// TIA Portal V17 export
// export: Created 2025-07-01T09:58:19.4161728Z, ExportSetting WithDefaults, DisplayName Totally Integrated Automation Portal, DisplayVersion V17 Update 8, DisplayName TIA Portal Openness, DisplayVersion V17 Update 8, DisplayName TIA Portal Version Control Interface, DisplayVersion V17, DisplayName SINAMICS Startdrive Advanced, DisplayVersion V17 SP2, DisplayName SINAMICS Startdrive G110M, G120, G120C, G120D, G120P, G115D, DisplayVersion V17 SP2, DisplayName SINAMICS Startdrive G130, G150, S120, S150, SINAMICS MV, S210, DisplayVersion V17 SP2, DisplayName STEP 7 Professional, DisplayVersion V17 Update 8, DisplayName SINUMERIK ONE STEP 7 Toolbox, DisplayVersion V17 Update 12, DisplayName SINUMERIK ONE PLC Basic Program Plus, DisplayVersion V17 Update 12, DisplayName SINUMERIK 840D sl STEP 7 Toolbox, DisplayVersion V17 Update 12, DisplayName STEP 7 Safety, DisplayVersion V17 Update 6, DisplayName WinCC Advanced, DisplayVersion V17 Update 8
FUNCTION_BLOCK "FB7001_SAFETY_DOOR"   // FB7001, LAD
{ S7_Optimized_Access := 'FALSE' }
AUTHOR : ETXETAR
VERSION : 1.0
// stored: AutoNumber false, IsIECCheckEnabled false, SetENOAutomatically false, UDAEnableTagReadback false
   VAR_INPUT
      OPTIONS_0 : Byte := 2#0000_0000;   // OPTIONS 0
      CLOSED_I : Bool;   // N.O / CLOSED INPUT
      LOCKED_I : Bool;   // N.O / LOCKED INPUT
      LOCK_CONDITIONS : Bool;   // LOCK CONDITIONS
      UNLOCK_PARTIAL_CONDITIONS : Bool;   // UNLOCK PARTIAL CONDITIONS
      HMI_REQ_LINE : Bool;   // HMI REQUEST LINE 1
      PANEL_LOCK_UNLOCK_PUSHBUTTON : Bool;   // PANEL LOCK UNLOCK PUSHBUTTON
      LOCK_AUTO_REQ : Bool;   // LOCK AUTO REQUEST
      UNLOCK_AUTO_REQ : Bool;   // UNLOCK AUTO REQUEST
      PNEUMATIC_DRIVE_UNBLOCKED : Bool;   // PNEUMATIC DRIVE 1 UNBLOCKED
   END_VAR
   VAR_OUTPUT
      NOT_CLOSED_AND_LOCKED_ALARM : Bool;   // NOT CLOSED AND LOCKED ALARM
      PNEUMATIC_DRIVE_NOT_UNBLOCKED_ALARM : Bool;   // PNEUMATIC DRIVE NOT UNBLOCKED ALARM
      NOT_OPEN_ALARM : Bool;   // NOT OPEN ALARM
      UNLOCK_REQUEST_SEOC_WRN : Bool;   // UNLOCK REQUEST SEOC WARNING
      NOT_CLOSED_WRN : Bool;   // NOT CLOSED WARNING
      HMI_MOTION_EXECUTABILITY_LEFT : Bool;   // HMI MOTION EXECUTABILITY LEFT
      HMI_MOTION_EXECUTABILITY_RIGHT : Bool;   // HMI MOTION EXECUTABILITY RIGHT
      HMI_MOTION_END_POS_LEFT : Bool;   // HMI MOTION END POSITION LEFT
      HMI_MOTION_END_POS_RIGHT : Bool;   // HMI MOTION END POSITION RIGHT
      HMI_MOTION_ACTIVE_LEFT : Bool;   // HMI MOTION ACTIVE LEFT
      HMI_MOTION_ACTIVE_RIGHT : Bool;   // HMI MOTION ACTIVE RIGHT
      UNLOCK : Bool;   // UNLOCK OUTPUT
      RED_LIGHT : Bool;   // RED LIGHT OUTPUT
      GREEN_LIGHT : Bool;   // GREEN LIGHT OUTPUT
   END_VAR
   VAR DB_SPECIFIC
      SAFETY_DOOR : "SAFETY_DOOR";
   END_VAR
   VAR_TEMP
      INPUTS_MASK : Byte;   // INPUTS_MASK
      O_BYTE_0 : Struct   // OPTIONS BYTE 0
         IMMEDIATE_STOP : Bool;   // IMMEDIATE STOP REACTION OPTION
         SEOC_WARNING : Bool;   // SEOC WARNING REACTION OPTION
         CLOSED_SENSOR : Bool;   // CLOSED SENSOR OPTION
         CIRCUIT_E2 : Bool;   // CIRCUIT E2 OPTION
         PNEUMATIC_DRIVE : Bool;   // PNEUMATIC DRIVE OPTION
         GANTRY_ROBOT_OK_TO_OPEN : Bool;   // GANTRY ROBOT OK TO OPEN SAFETY DOOR OPTION
         SPARE_6 : Bool;   // SPARE 6 OPTION
         SPARE_7 : Bool;   // SPARE 7 OPTION
      END_STRUCT;
      DB_NUMBER : DInt;   // DB NUMBER FOR ALARM AND HELP DECODING
   END_VAR
   // SAFETY_DOOR.TIMER_UNLOCK_PARTIAL_CONDITIONS.PT := T#250ms;
   // SAFETY_DOOR.TIMER_UNLOCK.PT := T#250ms;
   // SAFETY_DOOR.TIMER_PNEUMATIC_DRIVE_1_NOT_UNLOCKED.PT := T#2s;
   // SAFETY_DOOR.TIMER_NOT_OPEN.PT := T#3s;
   VAR_TEMP   // added for the SCL form of the ladder/FBD networks
      _w1 : Bool;
      _w2 : Bool;
   END_VAR
BEGIN

NETWORK
TITLE = READ INSTANCE DB
      L     DINO;
      +     10#800000;
      T     #DB_NUMBER;


REGION Network 2: OPTIONS
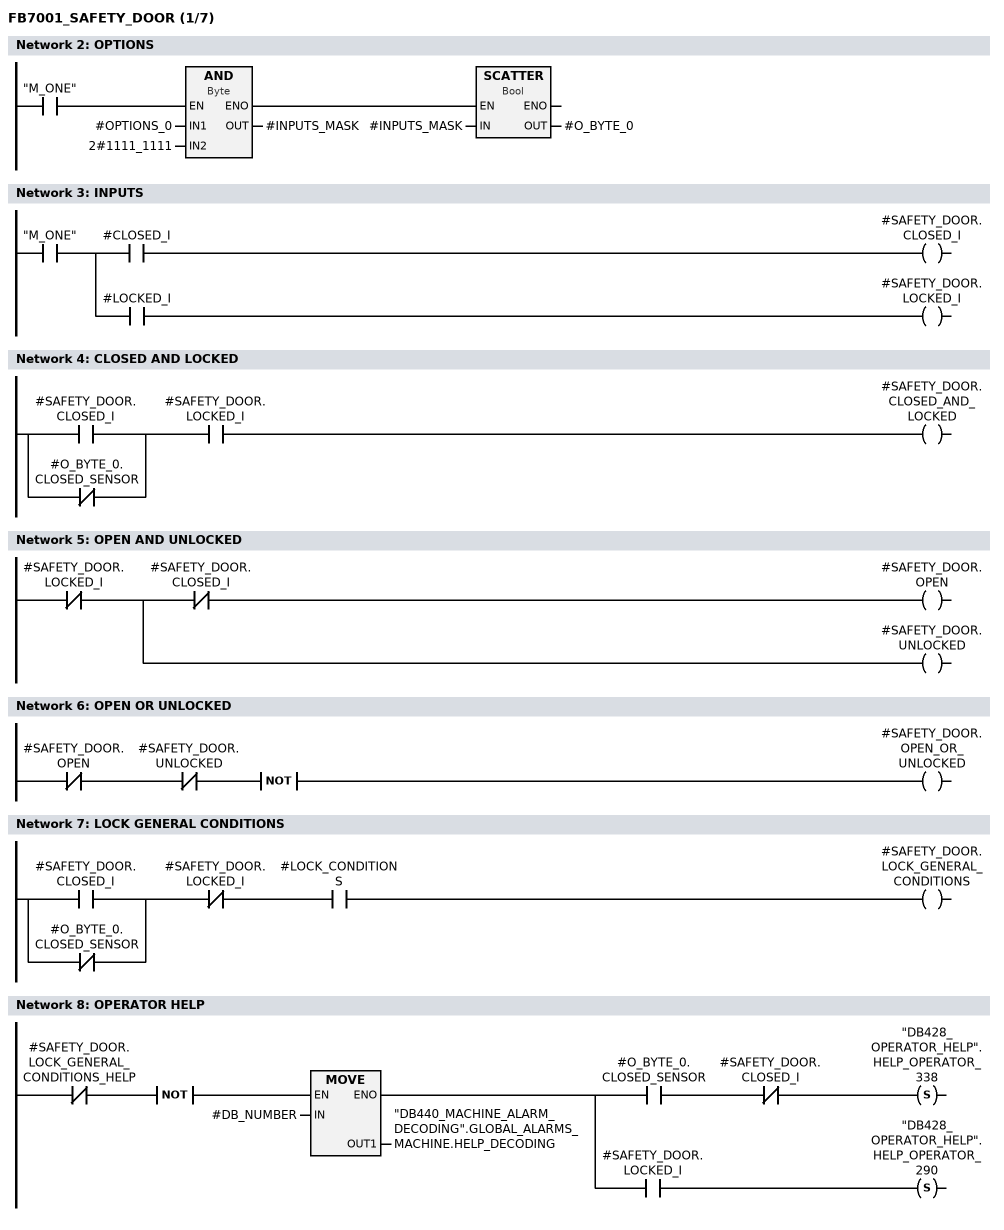
   RUNG wire#powerrail
      Contact( "M_ONE" )
      { S7_Templates := "SrcType := Byte"; S7_GenerateENO := "TRUE" } And(in1 := #OPTIONS_0, in2 := 2#1111_1111, out => #INPUTS_MASK)
      { S7_Templates := "[dest_type := Bool, src_type := Byte]" } SCATTER(IN := #INPUTS_MASK, OUT => #O_BYTE_0)
   END_RUNG
   // the same network as SCL:
   IF "M_ONE" THEN
       #INPUTS_MASK := #OPTIONS_0 AND 2#1111_1111;
       SCATTER(IN := #INPUTS_MASK, OUT => #O_BYTE_0);
   END_IF;
END_REGION

REGION Network 3: INPUTS
   RUNG wire#powerrail
      Contact( "M_ONE" )
      wire#w1
      Contact( #CLOSED_I )
      Coil( #SAFETY_DOOR.CLOSED_I )
   END_RUNG
   RUNG wire#w1
      Contact( #LOCKED_I )
      Coil( #SAFETY_DOOR.LOCKED_I )
   END_RUNG
   // the same network as SCL:
   #SAFETY_DOOR.CLOSED_I := "M_ONE" AND #CLOSED_I;
   #SAFETY_DOOR.LOCKED_I := "M_ONE" AND #LOCKED_I;
END_REGION

REGION Network 4: CLOSED AND LOCKED
   RUNG wire#powerrail
      Contact( #SAFETY_DOOR.CLOSED_I )
      wire#w1
      Contact( #SAFETY_DOOR.LOCKED_I )
      Coil( #SAFETY_DOOR.CLOSED_AND_LOCKED )
   END_RUNG
   RUNG wire#powerrail
      I_Contact( #O_BYTE_0.CLOSED_SENSOR )
   END_RUNG wire#w1
   // the same network as SCL:
   #SAFETY_DOOR.CLOSED_AND_LOCKED := (#SAFETY_DOOR.CLOSED_I OR NOT #O_BYTE_0.CLOSED_SENSOR) AND #SAFETY_DOOR.LOCKED_I;
END_REGION

REGION Network 5: OPEN AND UNLOCKED
   RUNG wire#powerrail
      I_Contact( #SAFETY_DOOR.LOCKED_I )
      wire#w1
      I_Contact( #SAFETY_DOOR.CLOSED_I )
      Coil( #SAFETY_DOOR.OPEN )
   END_RUNG
   RUNG wire#w1
      Coil( #SAFETY_DOOR.UNLOCKED )
   END_RUNG
   // the same network as SCL:
   #_w1 := NOT #SAFETY_DOOR.LOCKED_I;
   #SAFETY_DOOR.OPEN := #_w1 AND NOT #SAFETY_DOOR.CLOSED_I;
   #SAFETY_DOOR.UNLOCKED := #_w1;
END_REGION

REGION Network 6: OPEN OR UNLOCKED
   RUNG wire#powerrail
      I_Contact( #SAFETY_DOOR.OPEN )
      I_Contact( #SAFETY_DOOR.UNLOCKED )
      Not()
      Coil( #SAFETY_DOOR.OPEN_OR_UNLOCKED )
   END_RUNG
   // the same network as SCL:
   #SAFETY_DOOR.OPEN_OR_UNLOCKED := NOT (NOT #SAFETY_DOOR.OPEN AND NOT #SAFETY_DOOR.UNLOCKED);
END_REGION

REGION Network 7: LOCK GENERAL CONDITIONS
   RUNG wire#powerrail
      Contact( #SAFETY_DOOR.CLOSED_I )
      wire#w1
      I_Contact( #SAFETY_DOOR.LOCKED_I )
      Contact( #LOCK_CONDITIONS )
      Coil( #SAFETY_DOOR.LOCK_GENERAL_CONDITIONS )
   END_RUNG
   RUNG wire#powerrail
      I_Contact( #O_BYTE_0.CLOSED_SENSOR )
   END_RUNG wire#w1
   // the same network as SCL:
   #SAFETY_DOOR.LOCK_GENERAL_CONDITIONS := (#SAFETY_DOOR.CLOSED_I OR NOT #O_BYTE_0.CLOSED_SENSOR) AND NOT #SAFETY_DOOR.LOCKED_I AND #LOCK_CONDITIONS;
END_REGION

REGION Network 8: OPERATOR HELP
   RUNG wire#powerrail
      I_Contact( #SAFETY_DOOR.LOCK_GENERAL_CONDITIONS_HELP )
      Not()
      { S7_GenerateENO := "TRUE" } Move(in := #DB_NUMBER, out1 => "DB440_MACHINE_ALARM_DECODING".GLOBAL_ALARMS_MACHINE.HELP_DECODING)
      wire#w1
      Contact( #O_BYTE_0.CLOSED_SENSOR )
      I_Contact( #SAFETY_DOOR.CLOSED_I )
      S_Coil( "DB428_OPERATOR_HELP".HELP_OPERATOR_338 )
   END_RUNG
   RUNG wire#w1
      Contact( #SAFETY_DOOR.LOCKED_I )
      S_Coil( "DB428_OPERATOR_HELP".HELP_OPERATOR_290 )
   END_RUNG
   // the same network as SCL:
   // ENO of a box is taken as its EN; it also drops when the box reports an error
   #_w1 := NOT (NOT #SAFETY_DOOR.LOCK_GENERAL_CONDITIONS_HELP);
   IF #_w1 THEN "DB440_MACHINE_ALARM_DECODING".GLOBAL_ALARMS_MACHINE.HELP_DECODING := #DB_NUMBER; END_IF;
   IF #_w1 AND #O_BYTE_0.CLOSED_SENSOR AND NOT #SAFETY_DOOR.CLOSED_I THEN
       "DB428_OPERATOR_HELP".HELP_OPERATOR_338 := TRUE;
   END_IF;
   IF #_w1 AND #SAFETY_DOOR.LOCKED_I THEN "DB428_OPERATOR_HELP".HELP_OPERATOR_290 := TRUE; END_IF;
END_REGION

REGION Network 9: LOCK MANUAL REQUEST
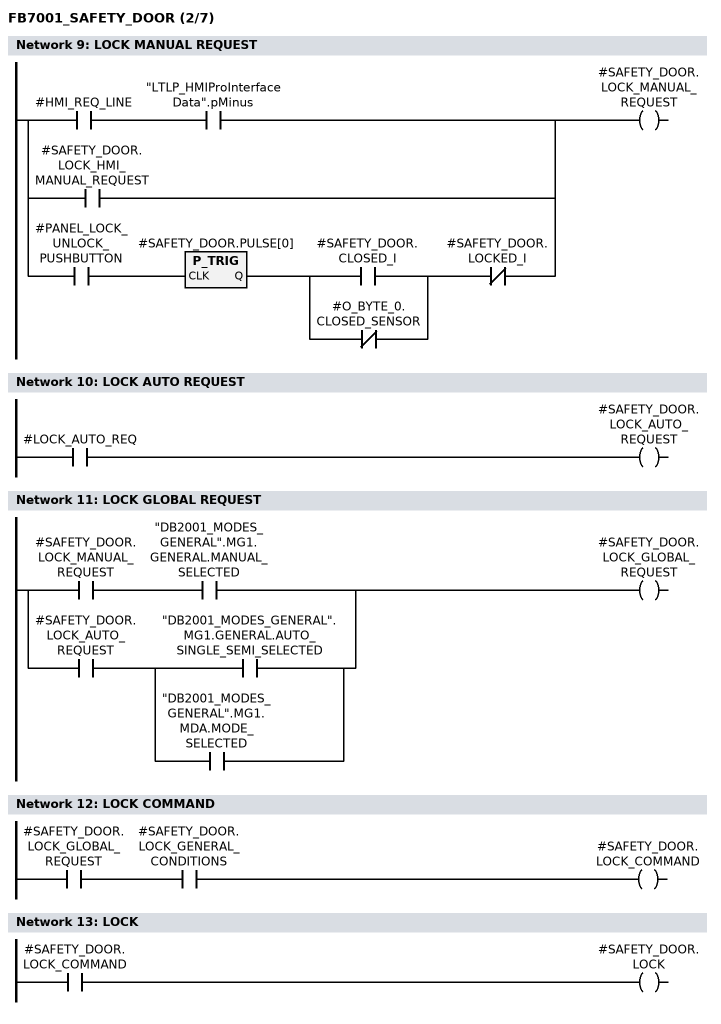
   RUNG wire#powerrail
      Contact( #HMI_REQ_LINE )
      Contact( "LTLP_HMIProInterfaceData".pMinus )
      wire#w1
      Coil( #SAFETY_DOOR.LOCK_MANUAL_REQUEST )
   END_RUNG
   RUNG wire#powerrail
      Contact( #SAFETY_DOOR.LOCK_HMI_MANUAL_REQUEST )
   END_RUNG wire#w1
   RUNG wire#powerrail
      Contact( #PANEL_LOCK_UNLOCK_PUSHBUTTON )
      P_Trig( #SAFETY_DOOR.PULSE[0] )
      wire#w2
      Contact( #SAFETY_DOOR.CLOSED_I )
      wire#w3
      I_Contact( #SAFETY_DOOR.LOCKED_I )
   END_RUNG wire#w1
   RUNG wire#w2
      I_Contact( #O_BYTE_0.CLOSED_SENSOR )
   END_RUNG wire#w3
   // the same network as SCL:
   #_w1 := #PANEL_LOCK_UNLOCK_PUSHBUTTON AND NOT #SAFETY_DOOR.PULSE[0];   // rising edge
   #SAFETY_DOOR.PULSE[0] := #PANEL_LOCK_UNLOCK_PUSHBUTTON;
   #SAFETY_DOOR.LOCK_MANUAL_REQUEST := (#HMI_REQ_LINE AND "LTLP_HMIProInterfaceData".pMinus) OR #SAFETY_DOOR.LOCK_HMI_MANUAL_REQUEST OR (#_w1 AND (#SAFETY_DOOR.CLOSED_I OR NOT #O_BYTE_0.CLOSED_SENSOR) AND NOT #SAFETY_DOOR.LOCKED_I);
END_REGION

REGION Network 10: LOCK AUTO REQUEST
   RUNG wire#powerrail
      Contact( #LOCK_AUTO_REQ )
      Coil( #SAFETY_DOOR.LOCK_AUTO_REQUEST )
   END_RUNG
   // the same network as SCL:
   #SAFETY_DOOR.LOCK_AUTO_REQUEST := #LOCK_AUTO_REQ;
END_REGION

REGION Network 11: LOCK GLOBAL REQUEST
   RUNG wire#powerrail
      Contact( #SAFETY_DOOR.LOCK_MANUAL_REQUEST )
      Contact( "DB2001_MODES_GENERAL".MG1.GENERAL.MANUAL_SELECTED )
      wire#w1
      Coil( #SAFETY_DOOR.LOCK_GLOBAL_REQUEST )
   END_RUNG
   RUNG wire#powerrail
      Contact( #SAFETY_DOOR.LOCK_AUTO_REQUEST )
      wire#w2
      Contact( "DB2001_MODES_GENERAL".MG1.GENERAL.AUTO_SINGLE_SEMI_SELECTED )
   END_RUNG wire#w1
   RUNG wire#w2
      Contact( "DB2001_MODES_GENERAL".MG1.MDA.MODE_SELECTED )
   END_RUNG wire#w1
   // the same network as SCL:
   #SAFETY_DOOR.LOCK_GLOBAL_REQUEST := (#SAFETY_DOOR.LOCK_MANUAL_REQUEST AND "DB2001_MODES_GENERAL".MG1.GENERAL.MANUAL_SELECTED) OR (#SAFETY_DOOR.LOCK_AUTO_REQUEST AND ("DB2001_MODES_GENERAL".MG1.GENERAL.AUTO_SINGLE_SEMI_SELECTED OR "DB2001_MODES_GENERAL".MG1.MDA.MODE_SELECTED));
END_REGION

REGION Network 12: LOCK COMMAND
   RUNG wire#powerrail
      Contact( #SAFETY_DOOR.LOCK_GLOBAL_REQUEST )
      Contact( #SAFETY_DOOR.LOCK_GENERAL_CONDITIONS )
      Coil( #SAFETY_DOOR.LOCK_COMMAND )
   END_RUNG
   // the same network as SCL:
   #SAFETY_DOOR.LOCK_COMMAND := #SAFETY_DOOR.LOCK_GLOBAL_REQUEST AND #SAFETY_DOOR.LOCK_GENERAL_CONDITIONS;
END_REGION

REGION Network 13: LOCK
   RUNG wire#powerrail
      Contact( #SAFETY_DOOR.LOCK_COMMAND )
      Coil( #SAFETY_DOOR.LOCK )
   END_RUNG
   // the same network as SCL:
   #SAFETY_DOOR.LOCK := #SAFETY_DOOR.LOCK_COMMAND;
END_REGION

REGION Network 14: UNLOCK PARTIAL CONDITIONS AUXILIARY
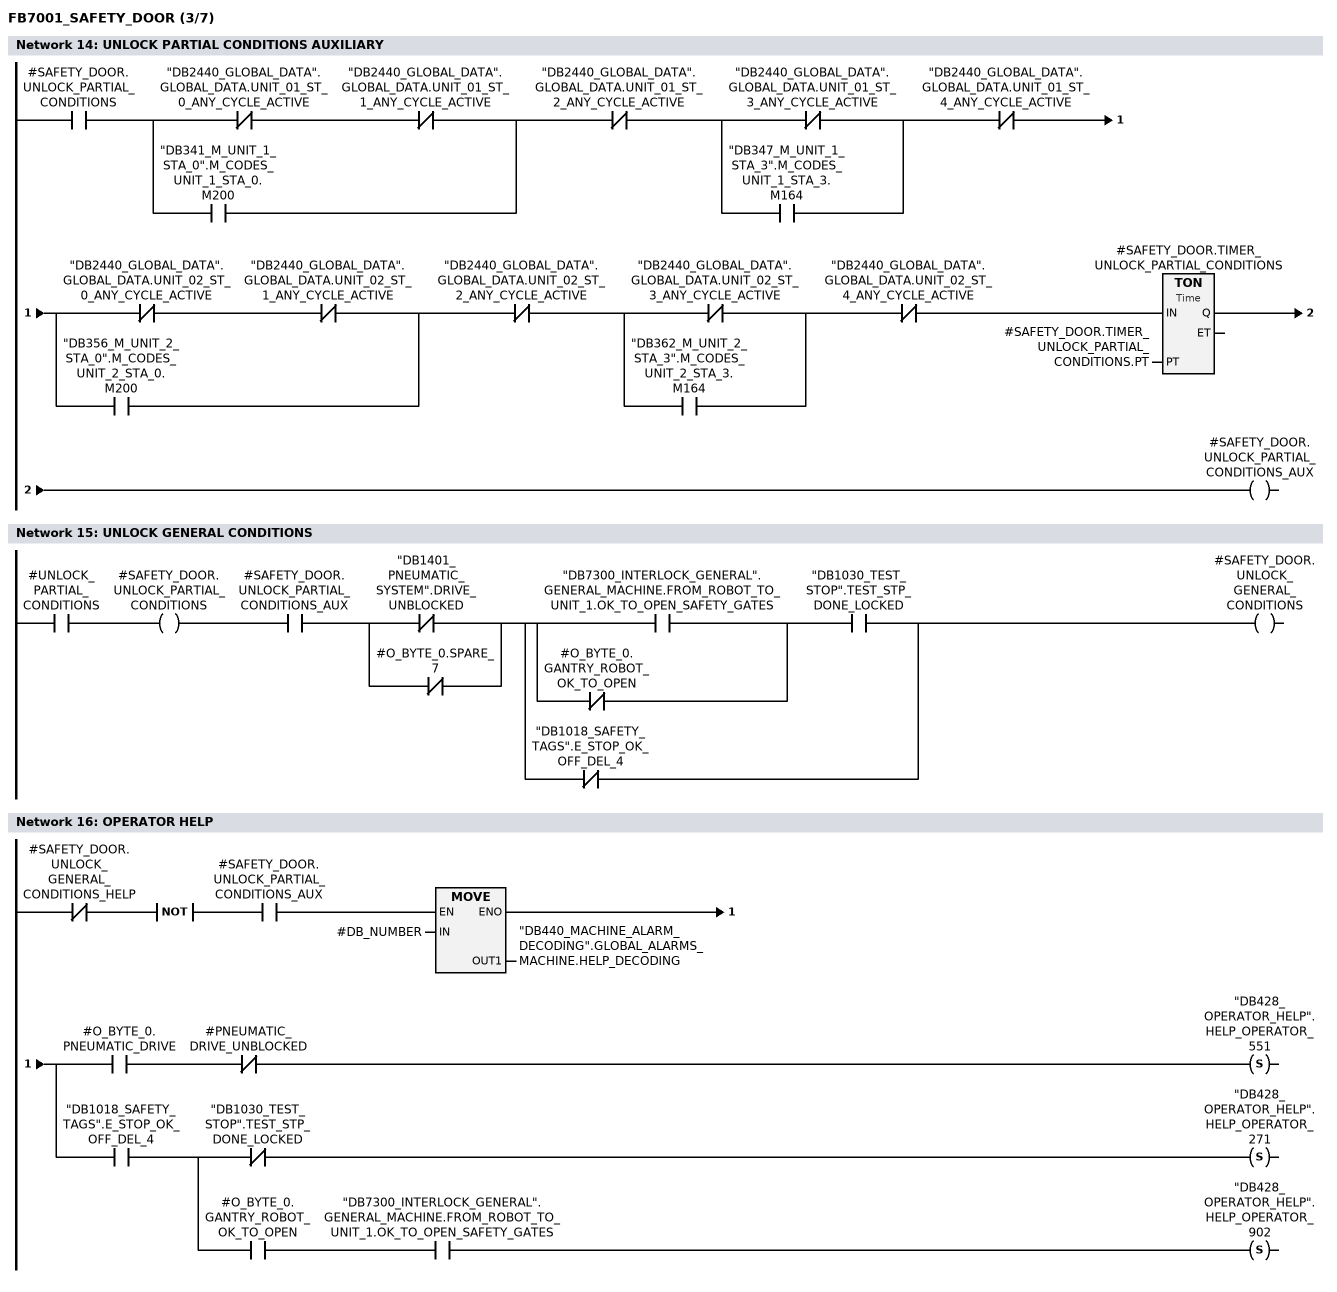
   RUNG wire#powerrail
      Contact( #SAFETY_DOOR.UNLOCK_PARTIAL_CONDITIONS )
      wire#w1
      I_Contact( "DB2440_GLOBAL_DATA".GLOBAL_DATA.UNIT_01_ST_0_ANY_CYCLE_ACTIVE )
      I_Contact( "DB2440_GLOBAL_DATA".GLOBAL_DATA.UNIT_01_ST_1_ANY_CYCLE_ACTIVE )
      wire#w2
      I_Contact( "DB2440_GLOBAL_DATA".GLOBAL_DATA.UNIT_01_ST_2_ANY_CYCLE_ACTIVE )
      wire#w3
      I_Contact( "DB2440_GLOBAL_DATA".GLOBAL_DATA.UNIT_01_ST_3_ANY_CYCLE_ACTIVE )
      wire#w4
      I_Contact( "DB2440_GLOBAL_DATA".GLOBAL_DATA.UNIT_01_ST_4_ANY_CYCLE_ACTIVE )
      wire#w5
      I_Contact( "DB2440_GLOBAL_DATA".GLOBAL_DATA.UNIT_02_ST_0_ANY_CYCLE_ACTIVE )
      I_Contact( "DB2440_GLOBAL_DATA".GLOBAL_DATA.UNIT_02_ST_1_ANY_CYCLE_ACTIVE )
      wire#w6
      I_Contact( "DB2440_GLOBAL_DATA".GLOBAL_DATA.UNIT_02_ST_2_ANY_CYCLE_ACTIVE )
      wire#w7
      I_Contact( "DB2440_GLOBAL_DATA".GLOBAL_DATA.UNIT_02_ST_3_ANY_CYCLE_ACTIVE )
      wire#w8
      I_Contact( "DB2440_GLOBAL_DATA".GLOBAL_DATA.UNIT_02_ST_4_ANY_CYCLE_ACTIVE )
      { S7_Templates := "time_type := Time" } #SAFETY_DOOR.TIMER_UNLOCK_PARTIAL_CONDITIONS.TON(pt := #SAFETY_DOOR.TIMER_UNLOCK_PARTIAL_CONDITIONS.PT, et =>)
      Coil( #SAFETY_DOOR.UNLOCK_PARTIAL_CONDITIONS_AUX )
   END_RUNG
   RUNG wire#w1
      Contact( "DB341_M_UNIT_1_STA_0".M_CODES_UNIT_1_STA_0.M200 )
   END_RUNG wire#w2
   RUNG wire#w3
      Contact( "DB347_M_UNIT_1_STA_3".M_CODES_UNIT_1_STA_3.M164 )
   END_RUNG wire#w4
   RUNG wire#w5
      Contact( "DB356_M_UNIT_2_STA_0".M_CODES_UNIT_2_STA_0.M200 )
   END_RUNG wire#w6
   RUNG wire#w7
      Contact( "DB362_M_UNIT_2_STA_3".M_CODES_UNIT_2_STA_3.M164 )
   END_RUNG wire#w8
   // the same network as SCL:
   #SAFETY_DOOR.TIMER_UNLOCK_PARTIAL_CONDITIONS.TON(IN := #SAFETY_DOOR.UNLOCK_PARTIAL_CONDITIONS AND ((NOT "DB2440_GLOBAL_DATA".GLOBAL_DATA.UNIT_01_ST_0_ANY_CYCLE_ACTIVE AND NOT "DB2440_GLOBAL_DATA".GLOBAL_DATA.UNIT_01_ST_1_ANY_CYCLE_ACTIVE) OR "DB341_M_UNIT_1_STA_0".M_CODES_UNIT_1_STA_0.M200) AND NOT "DB2440_GLOBAL_DATA".GLOBAL_DATA.UNIT_01_ST_2_ANY_CYCLE_ACTIVE AND (NOT "DB2440_GLOBAL_DATA".GLOBAL_DATA.UNIT_01_ST_3_ANY_CYCLE_ACTIVE OR "DB347_M_UNIT_1_STA_3".M_CODES_UNIT_1_STA_3.M164) AND NOT "DB2440_GLOBAL_DATA".GLOBAL_DATA.UNIT_01_ST_4_ANY_CYCLE_ACTIVE AND ((NOT "DB2440_GLOBAL_DATA".GLOBAL_DATA.UNIT_02_ST_0_ANY_CYCLE_ACTIVE AND NOT "DB2440_GLOBAL_DATA".GLOBAL_DATA.UNIT_02_ST_1_ANY_CYCLE_ACTIVE) OR "DB356_M_UNIT_2_STA_0".M_CODES_UNIT_2_STA_0.M200) AND NOT "DB2440_GLOBAL_DATA".GLOBAL_DATA.UNIT_02_ST_2_ANY_CYCLE_ACTIVE AND (NOT "DB2440_GLOBAL_DATA".GLOBAL_DATA.UNIT_02_ST_3_ANY_CYCLE_ACTIVE OR "DB362_M_UNIT_2_STA_3".M_CODES_UNIT_2_STA_3.M164) AND NOT "DB2440_GLOBAL_DATA".GLOBAL_DATA.UNIT_02_ST_4_ANY_CYCLE_ACTIVE,
                           PT := #SAFETY_DOOR.TIMER_UNLOCK_PARTIAL_CONDITIONS.PT);
   #SAFETY_DOOR.UNLOCK_PARTIAL_CONDITIONS_AUX := #SAFETY_DOOR.TIMER_UNLOCK_PARTIAL_CONDITIONS.Q;
END_REGION

REGION Network 15: UNLOCK GENERAL CONDITIONS
   RUNG wire#powerrail
      Contact( #UNLOCK_PARTIAL_CONDITIONS )
      Coil( #SAFETY_DOOR.UNLOCK_PARTIAL_CONDITIONS )
      Contact( #SAFETY_DOOR.UNLOCK_PARTIAL_CONDITIONS_AUX )
      wire#w1
      I_Contact( "DB1401_PNEUMATIC_SYSTEM".DRIVE_UNBLOCKED )
      wire#w2
      Contact( "DB7300_INTERLOCK_GENERAL".GENERAL_MACHINE.FROM_ROBOT_TO_UNIT_1.OK_TO_OPEN_SAFETY_GATES )
      wire#w3
      Contact( "DB1030_TEST_STOP".TEST_STP_DONE_LOCKED )
      wire#w4
      Coil( #SAFETY_DOOR.UNLOCK_GENERAL_CONDITIONS )
   END_RUNG
   RUNG wire#w1
      I_Contact( #O_BYTE_0.SPARE_7 )
   END_RUNG wire#w2
   RUNG wire#w2
      I_Contact( #O_BYTE_0.GANTRY_ROBOT_OK_TO_OPEN )
   END_RUNG wire#w3
   RUNG wire#w2
      I_Contact( "DB1018_SAFETY_TAGS".E_STOP_OK_OFF_DEL_4 )
   END_RUNG wire#w4
   // the same network as SCL:
   #SAFETY_DOOR.UNLOCK_PARTIAL_CONDITIONS := #UNLOCK_PARTIAL_CONDITIONS;
   #SAFETY_DOOR.UNLOCK_GENERAL_CONDITIONS := #UNLOCK_PARTIAL_CONDITIONS AND #SAFETY_DOOR.UNLOCK_PARTIAL_CONDITIONS_AUX AND (NOT "DB1401_PNEUMATIC_SYSTEM".DRIVE_UNBLOCKED OR NOT #O_BYTE_0.SPARE_7) AND ((("DB7300_INTERLOCK_GENERAL".GENERAL_MACHINE.FROM_ROBOT_TO_UNIT_1.OK_TO_OPEN_SAFETY_GATES OR NOT #O_BYTE_0.GANTRY_ROBOT_OK_TO_OPEN) AND "DB1030_TEST_STOP".TEST_STP_DONE_LOCKED) OR NOT "DB1018_SAFETY_TAGS".E_STOP_OK_OFF_DEL_4);
END_REGION

REGION Network 16: OPERATOR HELP
   RUNG wire#powerrail
      I_Contact( #SAFETY_DOOR.UNLOCK_GENERAL_CONDITIONS_HELP )
      Not()
      Contact( #SAFETY_DOOR.UNLOCK_PARTIAL_CONDITIONS_AUX )
      { S7_GenerateENO := "TRUE" } Move(in := #DB_NUMBER, out1 => "DB440_MACHINE_ALARM_DECODING".GLOBAL_ALARMS_MACHINE.HELP_DECODING)
      wire#w1
      Contact( #O_BYTE_0.PNEUMATIC_DRIVE )
      I_Contact( #PNEUMATIC_DRIVE_UNBLOCKED )
      S_Coil( "DB428_OPERATOR_HELP".HELP_OPERATOR_551 )
   END_RUNG
   RUNG wire#w1
      Contact( "DB1018_SAFETY_TAGS".E_STOP_OK_OFF_DEL_4 )
      wire#w2
      I_Contact( "DB1030_TEST_STOP".TEST_STP_DONE_LOCKED )
      S_Coil( "DB428_OPERATOR_HELP".HELP_OPERATOR_271 )
   END_RUNG
   RUNG wire#w2
      Contact( #O_BYTE_0.GANTRY_ROBOT_OK_TO_OPEN )
      Contact( "DB7300_INTERLOCK_GENERAL".GENERAL_MACHINE.FROM_ROBOT_TO_UNIT_1.OK_TO_OPEN_SAFETY_GATES )
      S_Coil( "DB428_OPERATOR_HELP".HELP_OPERATOR_902 )
   END_RUNG
   // the same network as SCL:
   // ENO of a box is taken as its EN; it also drops when the box reports an error
   #_w1 := NOT (NOT #SAFETY_DOOR.UNLOCK_GENERAL_CONDITIONS_HELP) AND #SAFETY_DOOR.UNLOCK_PARTIAL_CONDITIONS_AUX;
   IF #_w1 THEN "DB440_MACHINE_ALARM_DECODING".GLOBAL_ALARMS_MACHINE.HELP_DECODING := #DB_NUMBER; END_IF;
   IF #_w1 AND #O_BYTE_0.PNEUMATIC_DRIVE AND NOT #PNEUMATIC_DRIVE_UNBLOCKED THEN
       "DB428_OPERATOR_HELP".HELP_OPERATOR_551 := TRUE;
   END_IF;
   #_w2 := #_w1 AND "DB1018_SAFETY_TAGS".E_STOP_OK_OFF_DEL_4;
   IF #_w2 AND NOT "DB1030_TEST_STOP".TEST_STP_DONE_LOCKED THEN
       "DB428_OPERATOR_HELP".HELP_OPERATOR_271 := TRUE;
   END_IF;
   IF #_w2 AND #O_BYTE_0.GANTRY_ROBOT_OK_TO_OPEN AND "DB7300_INTERLOCK_GENERAL".GENERAL_MACHINE.FROM_ROBOT_TO_UNIT_1.OK_TO_OPEN_SAFETY_GATES THEN
       "DB428_OPERATOR_HELP".HELP_OPERATOR_902 := TRUE;
   END_IF;
END_REGION

REGION Network 17: UNLOCK MANUAL REQUEST
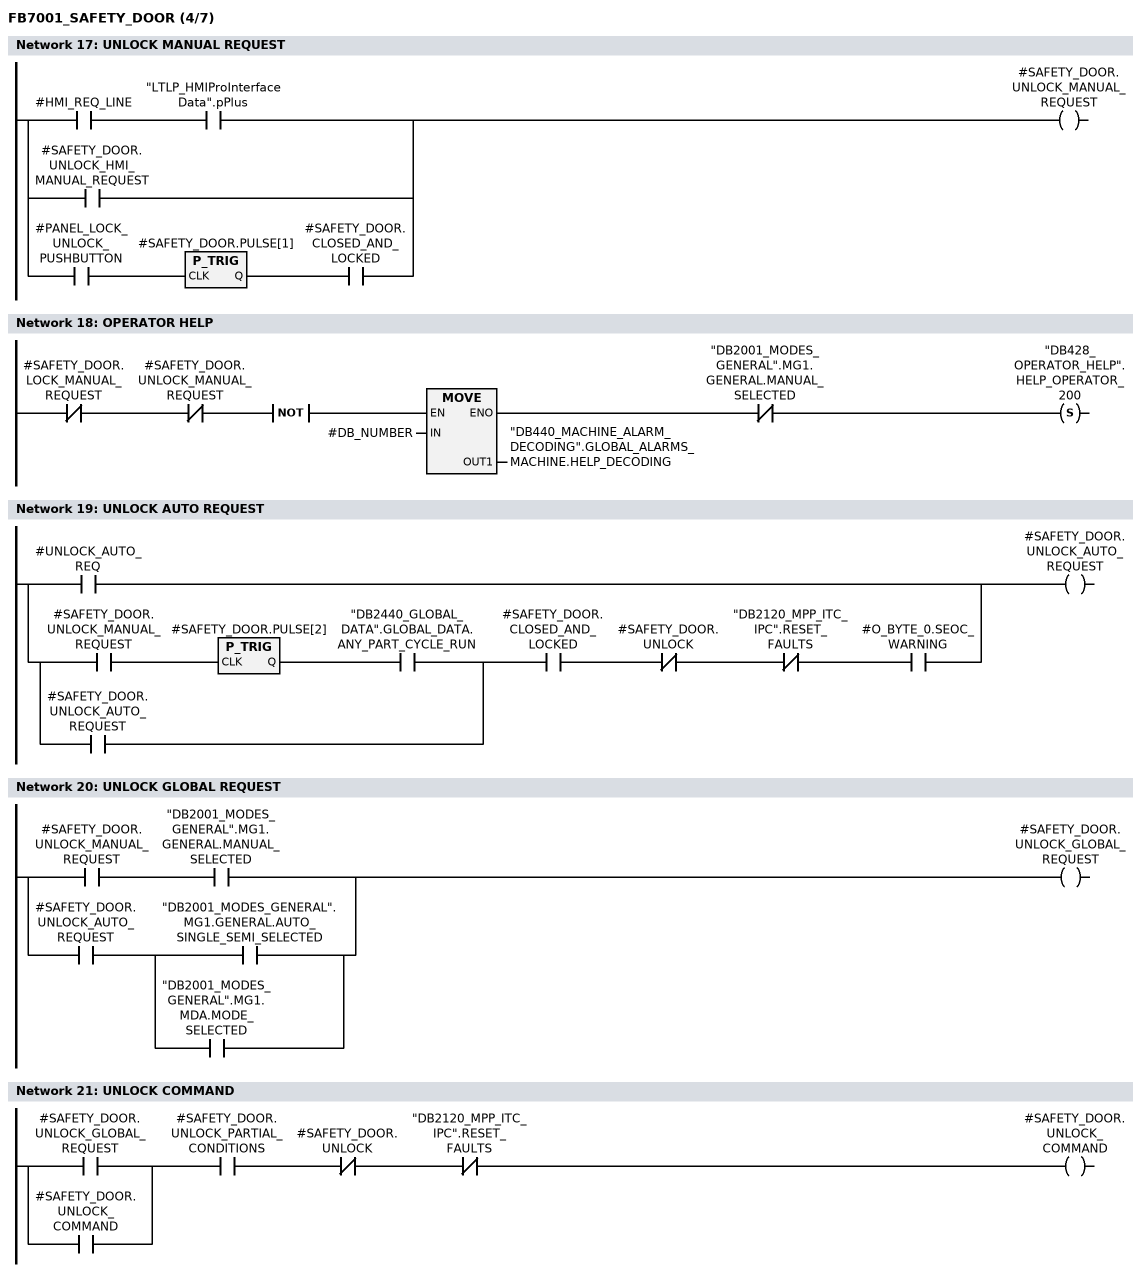
   RUNG wire#powerrail
      Contact( #HMI_REQ_LINE )
      Contact( "LTLP_HMIProInterfaceData".pPlus )
      wire#w1
      Coil( #SAFETY_DOOR.UNLOCK_MANUAL_REQUEST )
   END_RUNG
   RUNG wire#powerrail
      Contact( #SAFETY_DOOR.UNLOCK_HMI_MANUAL_REQUEST )
   END_RUNG wire#w1
   RUNG wire#powerrail
      Contact( #PANEL_LOCK_UNLOCK_PUSHBUTTON )
      P_Trig( #SAFETY_DOOR.PULSE[1] )
      Contact( #SAFETY_DOOR.CLOSED_AND_LOCKED )
   END_RUNG wire#w1
   // the same network as SCL:
   #_w1 := #PANEL_LOCK_UNLOCK_PUSHBUTTON AND NOT #SAFETY_DOOR.PULSE[1];   // rising edge
   #SAFETY_DOOR.PULSE[1] := #PANEL_LOCK_UNLOCK_PUSHBUTTON;
   #SAFETY_DOOR.UNLOCK_MANUAL_REQUEST := (#HMI_REQ_LINE AND "LTLP_HMIProInterfaceData".pPlus) OR #SAFETY_DOOR.UNLOCK_HMI_MANUAL_REQUEST OR (#_w1 AND #SAFETY_DOOR.CLOSED_AND_LOCKED);
END_REGION

REGION Network 18: OPERATOR HELP
   RUNG wire#powerrail
      I_Contact( #SAFETY_DOOR.LOCK_MANUAL_REQUEST )
      I_Contact( #SAFETY_DOOR.UNLOCK_MANUAL_REQUEST )
      Not()
      { S7_GenerateENO := "TRUE" } Move(in := #DB_NUMBER, out1 => "DB440_MACHINE_ALARM_DECODING".GLOBAL_ALARMS_MACHINE.HELP_DECODING)
      I_Contact( "DB2001_MODES_GENERAL".MG1.GENERAL.MANUAL_SELECTED )
      S_Coil( "DB428_OPERATOR_HELP".HELP_OPERATOR_200 )
   END_RUNG
   // the same network as SCL:
   // ENO of a box is taken as its EN; it also drops when the box reports an error
   #_w1 := NOT (NOT #SAFETY_DOOR.LOCK_MANUAL_REQUEST AND NOT #SAFETY_DOOR.UNLOCK_MANUAL_REQUEST);
   IF #_w1 THEN "DB440_MACHINE_ALARM_DECODING".GLOBAL_ALARMS_MACHINE.HELP_DECODING := #DB_NUMBER; END_IF;
   IF #_w1 AND NOT "DB2001_MODES_GENERAL".MG1.GENERAL.MANUAL_SELECTED THEN
       "DB428_OPERATOR_HELP".HELP_OPERATOR_200 := TRUE;
   END_IF;
END_REGION

REGION Network 19: UNLOCK AUTO REQUEST
   RUNG wire#powerrail
      Contact( #UNLOCK_AUTO_REQ )
      wire#w1
      Coil( #SAFETY_DOOR.UNLOCK_AUTO_REQUEST )
   END_RUNG
   RUNG wire#powerrail
      Contact( #SAFETY_DOOR.UNLOCK_MANUAL_REQUEST )
      P_Trig( #SAFETY_DOOR.PULSE[2] )
      Contact( "DB2440_GLOBAL_DATA".GLOBAL_DATA.ANY_PART_CYCLE_RUN )
      wire#w2
      Contact( #SAFETY_DOOR.CLOSED_AND_LOCKED )
      I_Contact( #SAFETY_DOOR.UNLOCK )
      I_Contact( "DB2120_MPP_ITC_IPC".RESET_FAULTS )
      Contact( #O_BYTE_0.SEOC_WARNING )
   END_RUNG wire#w1
   RUNG wire#powerrail
      Contact( #SAFETY_DOOR.UNLOCK_AUTO_REQUEST )
   END_RUNG wire#w2
   // the same network as SCL:
   #_w1 := #SAFETY_DOOR.UNLOCK_MANUAL_REQUEST AND NOT #SAFETY_DOOR.PULSE[2];   // rising edge
   #SAFETY_DOOR.PULSE[2] := #SAFETY_DOOR.UNLOCK_MANUAL_REQUEST;
   #SAFETY_DOOR.UNLOCK_AUTO_REQUEST := #UNLOCK_AUTO_REQ OR (((#_w1 AND "DB2440_GLOBAL_DATA".GLOBAL_DATA.ANY_PART_CYCLE_RUN) OR #SAFETY_DOOR.UNLOCK_AUTO_REQUEST) AND #SAFETY_DOOR.CLOSED_AND_LOCKED AND NOT #SAFETY_DOOR.UNLOCK AND NOT "DB2120_MPP_ITC_IPC".RESET_FAULTS AND #O_BYTE_0.SEOC_WARNING);
END_REGION

REGION Network 20: UNLOCK GLOBAL REQUEST
   RUNG wire#powerrail
      Contact( #SAFETY_DOOR.UNLOCK_MANUAL_REQUEST )
      Contact( "DB2001_MODES_GENERAL".MG1.GENERAL.MANUAL_SELECTED )
      wire#w1
      Coil( #SAFETY_DOOR.UNLOCK_GLOBAL_REQUEST )
   END_RUNG
   RUNG wire#powerrail
      Contact( #SAFETY_DOOR.UNLOCK_AUTO_REQUEST )
      wire#w2
      Contact( "DB2001_MODES_GENERAL".MG1.GENERAL.AUTO_SINGLE_SEMI_SELECTED )
   END_RUNG wire#w1
   RUNG wire#w2
      Contact( "DB2001_MODES_GENERAL".MG1.MDA.MODE_SELECTED )
   END_RUNG wire#w1
   // the same network as SCL:
   #SAFETY_DOOR.UNLOCK_GLOBAL_REQUEST := (#SAFETY_DOOR.UNLOCK_MANUAL_REQUEST AND "DB2001_MODES_GENERAL".MG1.GENERAL.MANUAL_SELECTED) OR (#SAFETY_DOOR.UNLOCK_AUTO_REQUEST AND ("DB2001_MODES_GENERAL".MG1.GENERAL.AUTO_SINGLE_SEMI_SELECTED OR "DB2001_MODES_GENERAL".MG1.MDA.MODE_SELECTED));
END_REGION

REGION Network 21: UNLOCK COMMAND
   RUNG wire#powerrail
      Contact( #SAFETY_DOOR.UNLOCK_GLOBAL_REQUEST )
      wire#w1
      Contact( #SAFETY_DOOR.UNLOCK_PARTIAL_CONDITIONS )
      I_Contact( #SAFETY_DOOR.UNLOCK )
      I_Contact( "DB2120_MPP_ITC_IPC".RESET_FAULTS )
      Coil( #SAFETY_DOOR.UNLOCK_COMMAND )
   END_RUNG
   RUNG wire#powerrail
      Contact( #SAFETY_DOOR.UNLOCK_COMMAND )
   END_RUNG wire#w1
   // the same network as SCL:
   #SAFETY_DOOR.UNLOCK_COMMAND := (#SAFETY_DOOR.UNLOCK_GLOBAL_REQUEST OR #SAFETY_DOOR.UNLOCK_COMMAND) AND #SAFETY_DOOR.UNLOCK_PARTIAL_CONDITIONS AND NOT #SAFETY_DOOR.UNLOCK AND NOT "DB2120_MPP_ITC_IPC".RESET_FAULTS;
END_REGION

REGION Network 22: UNLOCK
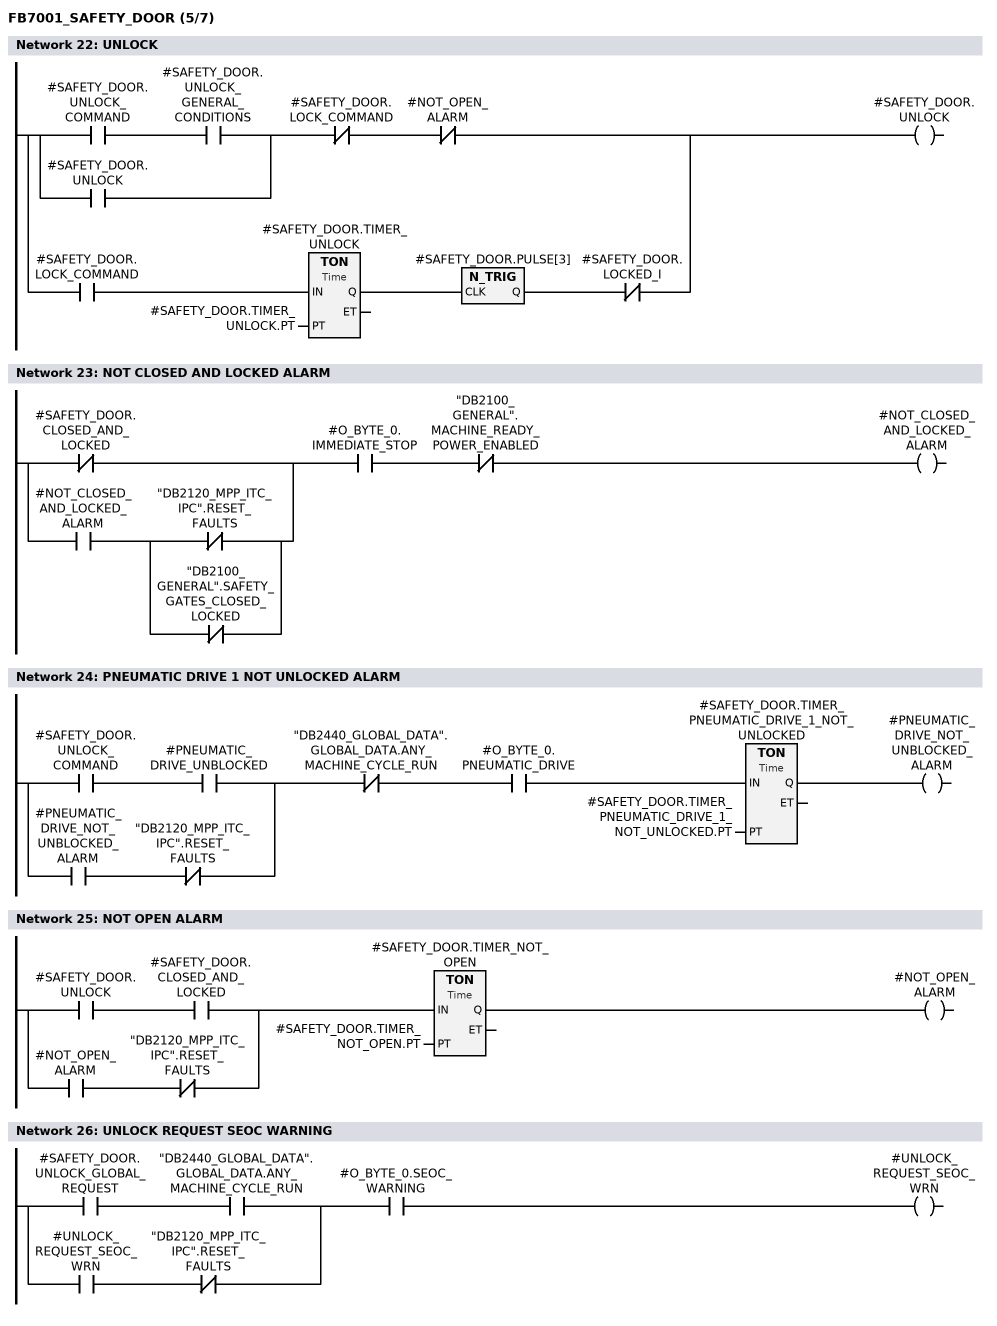
   RUNG wire#powerrail
      Contact( #SAFETY_DOOR.UNLOCK_COMMAND )
      Contact( #SAFETY_DOOR.UNLOCK_GENERAL_CONDITIONS )
      wire#w1
      I_Contact( #SAFETY_DOOR.LOCK_COMMAND )
      I_Contact( #NOT_OPEN_ALARM )
      wire#w2
      Coil( #SAFETY_DOOR.UNLOCK )
   END_RUNG
   RUNG wire#powerrail
      Contact( #SAFETY_DOOR.UNLOCK )
   END_RUNG wire#w1
   RUNG wire#powerrail
      Contact( #SAFETY_DOOR.LOCK_COMMAND )
      { S7_Templates := "time_type := Time" } #SAFETY_DOOR.TIMER_UNLOCK.TON(pt := #SAFETY_DOOR.TIMER_UNLOCK.PT, et =>)
      N_Trig( #SAFETY_DOOR.PULSE[3] )
      I_Contact( #SAFETY_DOOR.LOCKED_I )
   END_RUNG wire#w2
   // the same network as SCL:
   #SAFETY_DOOR.TIMER_UNLOCK.TON(IN := #SAFETY_DOOR.LOCK_COMMAND, PT := #SAFETY_DOOR.TIMER_UNLOCK.PT);
   #_w1 := NOT #SAFETY_DOOR.TIMER_UNLOCK.Q AND #SAFETY_DOOR.PULSE[3];   // falling edge
   #SAFETY_DOOR.PULSE[3] := #SAFETY_DOOR.TIMER_UNLOCK.Q;
   #SAFETY_DOOR.UNLOCK := (((#SAFETY_DOOR.UNLOCK_COMMAND AND #SAFETY_DOOR.UNLOCK_GENERAL_CONDITIONS) OR #SAFETY_DOOR.UNLOCK) AND NOT #SAFETY_DOOR.LOCK_COMMAND AND NOT #NOT_OPEN_ALARM) OR (#_w1 AND NOT #SAFETY_DOOR.LOCKED_I);
END_REGION

REGION Network 23: NOT CLOSED AND LOCKED ALARM
   RUNG wire#powerrail
      I_Contact( #SAFETY_DOOR.CLOSED_AND_LOCKED )
      wire#w1
      Contact( #O_BYTE_0.IMMEDIATE_STOP )
      I_Contact( "DB2100_GENERAL".MACHINE_READY_POWER_ENABLED )
      Coil( #NOT_CLOSED_AND_LOCKED_ALARM )
   END_RUNG
   RUNG wire#powerrail
      Contact( #NOT_CLOSED_AND_LOCKED_ALARM )
      wire#w2
      I_Contact( "DB2120_MPP_ITC_IPC".RESET_FAULTS )
   END_RUNG wire#w1
   RUNG wire#w2
      I_Contact( "DB2100_GENERAL".SAFETY_GATES_CLOSED_LOCKED )
   END_RUNG wire#w1
   // the same network as SCL:
   #NOT_CLOSED_AND_LOCKED_ALARM := (NOT #SAFETY_DOOR.CLOSED_AND_LOCKED OR (#NOT_CLOSED_AND_LOCKED_ALARM AND (NOT "DB2120_MPP_ITC_IPC".RESET_FAULTS OR NOT "DB2100_GENERAL".SAFETY_GATES_CLOSED_LOCKED))) AND #O_BYTE_0.IMMEDIATE_STOP AND NOT "DB2100_GENERAL".MACHINE_READY_POWER_ENABLED;
END_REGION

REGION Network 24: PNEUMATIC DRIVE 1 NOT UNLOCKED ALARM
   RUNG wire#powerrail
      Contact( #SAFETY_DOOR.UNLOCK_COMMAND )
      Contact( #PNEUMATIC_DRIVE_UNBLOCKED )
      wire#w1
      I_Contact( "DB2440_GLOBAL_DATA".GLOBAL_DATA.ANY_MACHINE_CYCLE_RUN )
      Contact( #O_BYTE_0.PNEUMATIC_DRIVE )
      { S7_Templates := "time_type := Time" } #SAFETY_DOOR.TIMER_PNEUMATIC_DRIVE_1_NOT_UNLOCKED.TON(pt := #SAFETY_DOOR.TIMER_PNEUMATIC_DRIVE_1_NOT_UNLOCKED.PT, et =>)
      Coil( #PNEUMATIC_DRIVE_NOT_UNBLOCKED_ALARM )
   END_RUNG
   RUNG wire#powerrail
      Contact( #PNEUMATIC_DRIVE_NOT_UNBLOCKED_ALARM )
      I_Contact( "DB2120_MPP_ITC_IPC".RESET_FAULTS )
   END_RUNG wire#w1
   // the same network as SCL:
   #SAFETY_DOOR.TIMER_PNEUMATIC_DRIVE_1_NOT_UNLOCKED.TON(IN := ((#SAFETY_DOOR.UNLOCK_COMMAND AND #PNEUMATIC_DRIVE_UNBLOCKED) OR (#PNEUMATIC_DRIVE_NOT_UNBLOCKED_ALARM AND NOT "DB2120_MPP_ITC_IPC".RESET_FAULTS)) AND NOT "DB2440_GLOBAL_DATA".GLOBAL_DATA.ANY_MACHINE_CYCLE_RUN AND #O_BYTE_0.PNEUMATIC_DRIVE,
                           PT := #SAFETY_DOOR.TIMER_PNEUMATIC_DRIVE_1_NOT_UNLOCKED.PT);
   #PNEUMATIC_DRIVE_NOT_UNBLOCKED_ALARM := #SAFETY_DOOR.TIMER_PNEUMATIC_DRIVE_1_NOT_UNLOCKED.Q;
END_REGION

REGION Network 25: NOT OPEN ALARM
   RUNG wire#powerrail
      Contact( #SAFETY_DOOR.UNLOCK )
      Contact( #SAFETY_DOOR.CLOSED_AND_LOCKED )
      wire#w1
      { S7_Templates := "time_type := Time" } #SAFETY_DOOR.TIMER_NOT_OPEN.TON(pt := #SAFETY_DOOR.TIMER_NOT_OPEN.PT, et =>)
      Coil( #NOT_OPEN_ALARM )
   END_RUNG
   RUNG wire#powerrail
      Contact( #NOT_OPEN_ALARM )
      I_Contact( "DB2120_MPP_ITC_IPC".RESET_FAULTS )
   END_RUNG wire#w1
   // the same network as SCL:
   #SAFETY_DOOR.TIMER_NOT_OPEN.TON(IN := (#SAFETY_DOOR.UNLOCK AND #SAFETY_DOOR.CLOSED_AND_LOCKED) OR (#NOT_OPEN_ALARM AND NOT "DB2120_MPP_ITC_IPC".RESET_FAULTS),
                           PT := #SAFETY_DOOR.TIMER_NOT_OPEN.PT);
   #NOT_OPEN_ALARM := #SAFETY_DOOR.TIMER_NOT_OPEN.Q;
END_REGION

REGION Network 26: UNLOCK REQUEST SEOC WARNING
   RUNG wire#powerrail
      Contact( #SAFETY_DOOR.UNLOCK_GLOBAL_REQUEST )
      Contact( "DB2440_GLOBAL_DATA".GLOBAL_DATA.ANY_MACHINE_CYCLE_RUN )
      wire#w1
      Contact( #O_BYTE_0.SEOC_WARNING )
      Coil( #UNLOCK_REQUEST_SEOC_WRN )
   END_RUNG
   RUNG wire#powerrail
      Contact( #UNLOCK_REQUEST_SEOC_WRN )
      I_Contact( "DB2120_MPP_ITC_IPC".RESET_FAULTS )
   END_RUNG wire#w1
   // the same network as SCL:
   #UNLOCK_REQUEST_SEOC_WRN := ((#SAFETY_DOOR.UNLOCK_GLOBAL_REQUEST AND "DB2440_GLOBAL_DATA".GLOBAL_DATA.ANY_MACHINE_CYCLE_RUN) OR (#UNLOCK_REQUEST_SEOC_WRN AND NOT "DB2120_MPP_ITC_IPC".RESET_FAULTS)) AND #O_BYTE_0.SEOC_WARNING;
END_REGION

REGION Network 27: IMMEDIATE STOP ALARMS
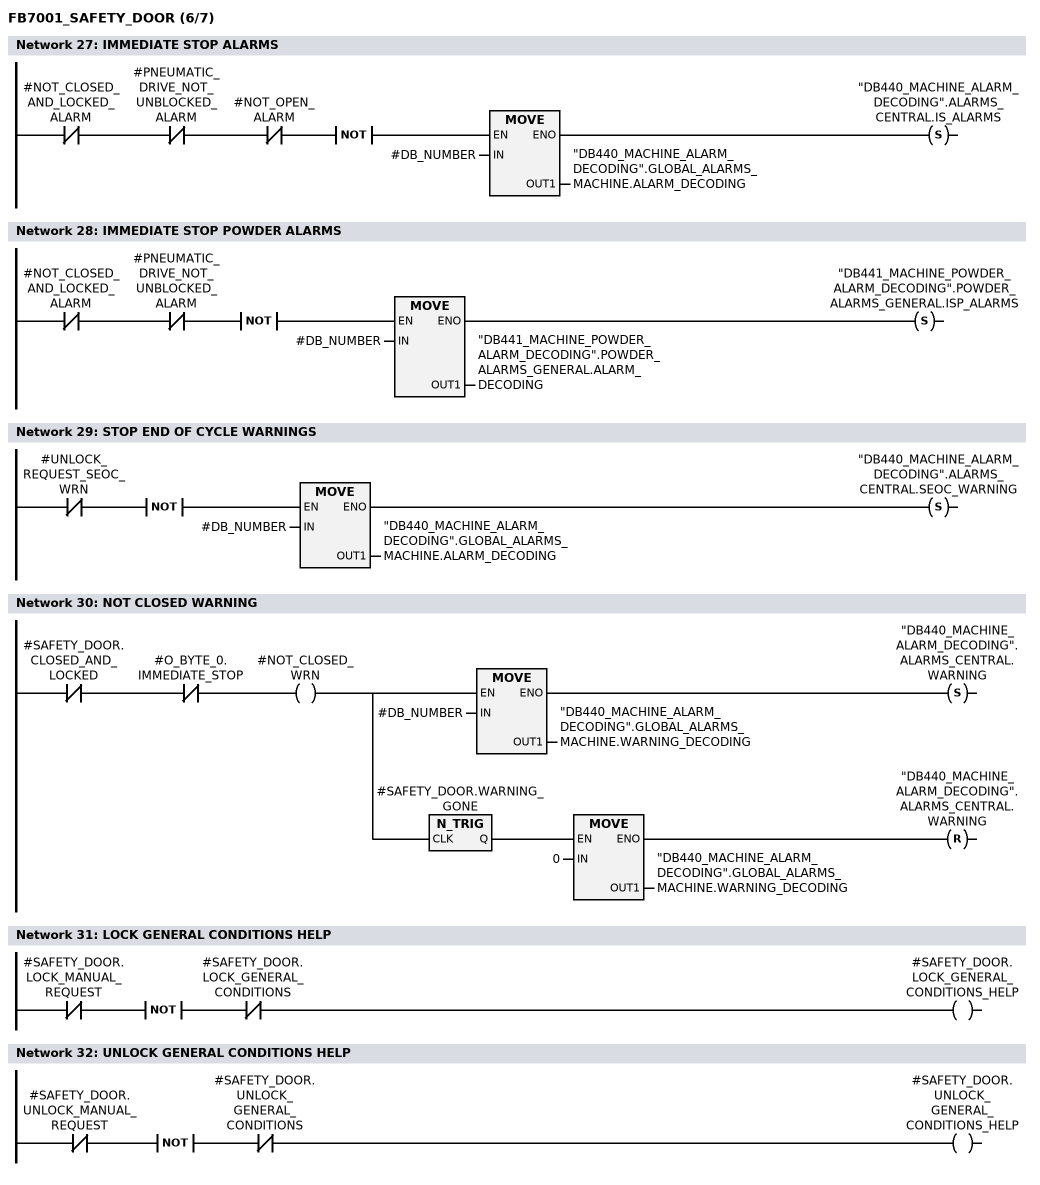
   RUNG wire#powerrail
      I_Contact( #NOT_CLOSED_AND_LOCKED_ALARM )
      I_Contact( #PNEUMATIC_DRIVE_NOT_UNBLOCKED_ALARM )
      I_Contact( #NOT_OPEN_ALARM )
      Not()
      { S7_GenerateENO := "TRUE" } Move(in := #DB_NUMBER, out1 => "DB440_MACHINE_ALARM_DECODING".GLOBAL_ALARMS_MACHINE.ALARM_DECODING)
      S_Coil( "DB440_MACHINE_ALARM_DECODING".ALARMS_CENTRAL.IS_ALARMS )
   END_RUNG
   // the same network as SCL:
   // ENO of a box is taken as its EN; it also drops when the box reports an error
   IF NOT (NOT #NOT_CLOSED_AND_LOCKED_ALARM AND NOT #PNEUMATIC_DRIVE_NOT_UNBLOCKED_ALARM AND NOT #NOT_OPEN_ALARM) THEN
       "DB440_MACHINE_ALARM_DECODING".GLOBAL_ALARMS_MACHINE.ALARM_DECODING := #DB_NUMBER;
       "DB440_MACHINE_ALARM_DECODING".ALARMS_CENTRAL.IS_ALARMS := TRUE;
   END_IF;
END_REGION

REGION Network 28: IMMEDIATE STOP POWDER ALARMS
   RUNG wire#powerrail
      I_Contact( #NOT_CLOSED_AND_LOCKED_ALARM )
      I_Contact( #PNEUMATIC_DRIVE_NOT_UNBLOCKED_ALARM )
      Not()
      { S7_GenerateENO := "TRUE" } Move(in := #DB_NUMBER, out1 => "DB441_MACHINE_POWDER_ALARM_DECODING".POWDER_ALARMS_GENERAL.ALARM_DECODING)
      S_Coil( "DB441_MACHINE_POWDER_ALARM_DECODING".POWDER_ALARMS_GENERAL.ISP_ALARMS )
   END_RUNG
   // the same network as SCL:
   // ENO of a box is taken as its EN; it also drops when the box reports an error
   IF NOT (NOT #NOT_CLOSED_AND_LOCKED_ALARM AND NOT #PNEUMATIC_DRIVE_NOT_UNBLOCKED_ALARM) THEN
       "DB441_MACHINE_POWDER_ALARM_DECODING".POWDER_ALARMS_GENERAL.ALARM_DECODING := #DB_NUMBER;
       "DB441_MACHINE_POWDER_ALARM_DECODING".POWDER_ALARMS_GENERAL.ISP_ALARMS := TRUE;
   END_IF;
END_REGION

REGION Network 29: STOP END OF CYCLE WARNINGS
   RUNG wire#powerrail
      I_Contact( #UNLOCK_REQUEST_SEOC_WRN )
      Not()
      { S7_GenerateENO := "TRUE" } Move(in := #DB_NUMBER, out1 => "DB440_MACHINE_ALARM_DECODING".GLOBAL_ALARMS_MACHINE.ALARM_DECODING)
      S_Coil( "DB440_MACHINE_ALARM_DECODING".ALARMS_CENTRAL.SEOC_WARNING )
   END_RUNG
   // the same network as SCL:
   // ENO of a box is taken as its EN; it also drops when the box reports an error
   IF NOT (NOT #UNLOCK_REQUEST_SEOC_WRN) THEN
       "DB440_MACHINE_ALARM_DECODING".GLOBAL_ALARMS_MACHINE.ALARM_DECODING := #DB_NUMBER;
       "DB440_MACHINE_ALARM_DECODING".ALARMS_CENTRAL.SEOC_WARNING := TRUE;
   END_IF;
END_REGION

REGION Network 30: NOT CLOSED WARNING
   RUNG wire#powerrail
      I_Contact( #SAFETY_DOOR.CLOSED_AND_LOCKED )
      I_Contact( #O_BYTE_0.IMMEDIATE_STOP )
      Coil( #NOT_CLOSED_WRN )
      wire#w1
      { S7_GenerateENO := "TRUE" } Move(in := #DB_NUMBER, out1 => "DB440_MACHINE_ALARM_DECODING".GLOBAL_ALARMS_MACHINE.WARNING_DECODING)
      S_Coil( "DB440_MACHINE_ALARM_DECODING".ALARMS_CENTRAL.WARNING )
   END_RUNG
   RUNG wire#w1
      N_Trig( #SAFETY_DOOR.WARNING_GONE )
      { S7_GenerateENO := "TRUE" } Move(in := 0, out1 => "DB440_MACHINE_ALARM_DECODING".GLOBAL_ALARMS_MACHINE.WARNING_DECODING)
      R_Coil( "DB440_MACHINE_ALARM_DECODING".ALARMS_CENTRAL.WARNING )
   END_RUNG
   // the same network as SCL:
   // ENO of a box is taken as its EN; it also drops when the box reports an error
   #NOT_CLOSED_WRN := NOT #SAFETY_DOOR.CLOSED_AND_LOCKED AND NOT #O_BYTE_0.IMMEDIATE_STOP;
   IF #NOT_CLOSED_WRN THEN
       "DB440_MACHINE_ALARM_DECODING".GLOBAL_ALARMS_MACHINE.WARNING_DECODING := #DB_NUMBER;
       "DB440_MACHINE_ALARM_DECODING".ALARMS_CENTRAL.WARNING := TRUE;
   END_IF;
   #_w1 := NOT #NOT_CLOSED_WRN AND #SAFETY_DOOR.WARNING_GONE;   // falling edge
   #SAFETY_DOOR.WARNING_GONE := #NOT_CLOSED_WRN;
   IF #_w1 THEN
       "DB440_MACHINE_ALARM_DECODING".GLOBAL_ALARMS_MACHINE.WARNING_DECODING := 0;
       "DB440_MACHINE_ALARM_DECODING".ALARMS_CENTRAL.WARNING := FALSE;
   END_IF;
END_REGION

REGION Network 31: LOCK GENERAL CONDITIONS HELP
   RUNG wire#powerrail
      I_Contact( #SAFETY_DOOR.LOCK_MANUAL_REQUEST )
      Not()
      I_Contact( #SAFETY_DOOR.LOCK_GENERAL_CONDITIONS )
      Coil( #SAFETY_DOOR.LOCK_GENERAL_CONDITIONS_HELP )
   END_RUNG
   // the same network as SCL:
   #SAFETY_DOOR.LOCK_GENERAL_CONDITIONS_HELP := NOT (NOT #SAFETY_DOOR.LOCK_MANUAL_REQUEST) AND NOT #SAFETY_DOOR.LOCK_GENERAL_CONDITIONS;
END_REGION

REGION Network 32: UNLOCK GENERAL CONDITIONS HELP
   RUNG wire#powerrail
      I_Contact( #SAFETY_DOOR.UNLOCK_MANUAL_REQUEST )
      Not()
      I_Contact( #SAFETY_DOOR.UNLOCK_GENERAL_CONDITIONS )
      Coil( #SAFETY_DOOR.UNLOCK_GENERAL_CONDITIONS_HELP )
   END_RUNG
   // the same network as SCL:
   #SAFETY_DOOR.UNLOCK_GENERAL_CONDITIONS_HELP := NOT (NOT #SAFETY_DOOR.UNLOCK_MANUAL_REQUEST) AND NOT #SAFETY_DOOR.UNLOCK_GENERAL_CONDITIONS;
END_REGION

REGION Network 33: HMI STATUS
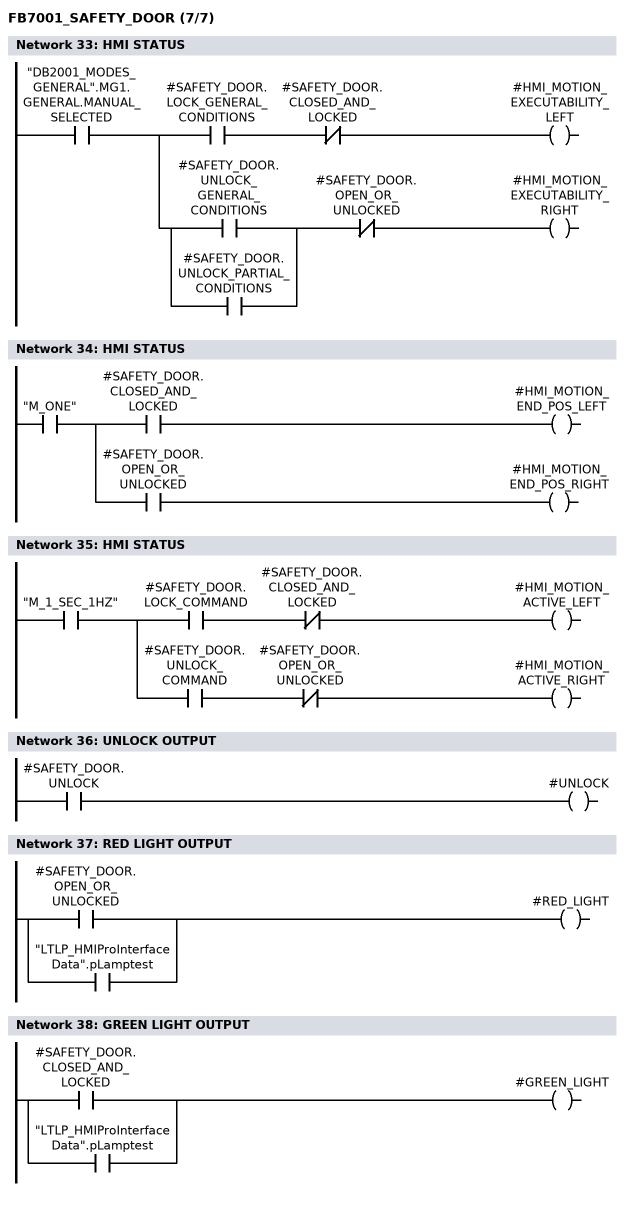
   RUNG wire#powerrail
      Contact( "DB2001_MODES_GENERAL".MG1.GENERAL.MANUAL_SELECTED )
      wire#w1
      Contact( #SAFETY_DOOR.LOCK_GENERAL_CONDITIONS )
      I_Contact( #SAFETY_DOOR.CLOSED_AND_LOCKED )
      Coil( #HMI_MOTION_EXECUTABILITY_LEFT )
   END_RUNG
   RUNG wire#w1
      Contact( #SAFETY_DOOR.UNLOCK_GENERAL_CONDITIONS )
      wire#w2
      I_Contact( #SAFETY_DOOR.OPEN_OR_UNLOCKED )
      Coil( #HMI_MOTION_EXECUTABILITY_RIGHT )
   END_RUNG
   RUNG wire#w1
      Contact( #SAFETY_DOOR.UNLOCK_PARTIAL_CONDITIONS )
   END_RUNG wire#w2
   // the same network as SCL:
   #HMI_MOTION_EXECUTABILITY_LEFT := "DB2001_MODES_GENERAL".MG1.GENERAL.MANUAL_SELECTED AND #SAFETY_DOOR.LOCK_GENERAL_CONDITIONS AND NOT #SAFETY_DOOR.CLOSED_AND_LOCKED;
   #HMI_MOTION_EXECUTABILITY_RIGHT := "DB2001_MODES_GENERAL".MG1.GENERAL.MANUAL_SELECTED AND (#SAFETY_DOOR.UNLOCK_GENERAL_CONDITIONS OR #SAFETY_DOOR.UNLOCK_PARTIAL_CONDITIONS) AND NOT #SAFETY_DOOR.OPEN_OR_UNLOCKED;
END_REGION

REGION Network 34: HMI STATUS
   RUNG wire#powerrail
      Contact( "M_ONE" )
      wire#w1
      Contact( #SAFETY_DOOR.CLOSED_AND_LOCKED )
      Coil( #HMI_MOTION_END_POS_LEFT )
   END_RUNG
   RUNG wire#w1
      Contact( #SAFETY_DOOR.OPEN_OR_UNLOCKED )
      Coil( #HMI_MOTION_END_POS_RIGHT )
   END_RUNG
   // the same network as SCL:
   #HMI_MOTION_END_POS_LEFT := "M_ONE" AND #SAFETY_DOOR.CLOSED_AND_LOCKED;
   #HMI_MOTION_END_POS_RIGHT := "M_ONE" AND #SAFETY_DOOR.OPEN_OR_UNLOCKED;
END_REGION

REGION Network 35: HMI STATUS
   RUNG wire#powerrail
      Contact( "M_1_SEC_1HZ" )
      wire#w1
      Contact( #SAFETY_DOOR.LOCK_COMMAND )
      I_Contact( #SAFETY_DOOR.CLOSED_AND_LOCKED )
      Coil( #HMI_MOTION_ACTIVE_LEFT )
   END_RUNG
   RUNG wire#w1
      Contact( #SAFETY_DOOR.UNLOCK_COMMAND )
      I_Contact( #SAFETY_DOOR.OPEN_OR_UNLOCKED )
      Coil( #HMI_MOTION_ACTIVE_RIGHT )
   END_RUNG
   // the same network as SCL:
   #HMI_MOTION_ACTIVE_LEFT := "M_1_SEC_1HZ" AND #SAFETY_DOOR.LOCK_COMMAND AND NOT #SAFETY_DOOR.CLOSED_AND_LOCKED;
   #HMI_MOTION_ACTIVE_RIGHT := "M_1_SEC_1HZ" AND #SAFETY_DOOR.UNLOCK_COMMAND AND NOT #SAFETY_DOOR.OPEN_OR_UNLOCKED;
END_REGION

REGION Network 36: UNLOCK OUTPUT
   RUNG wire#powerrail
      Contact( #SAFETY_DOOR.UNLOCK )
      Coil( #UNLOCK )
   END_RUNG
   // the same network as SCL:
   #UNLOCK := #SAFETY_DOOR.UNLOCK;
END_REGION

REGION Network 37: RED LIGHT OUTPUT
   RUNG wire#powerrail
      Contact( #SAFETY_DOOR.OPEN_OR_UNLOCKED )
      wire#w1
      Coil( #RED_LIGHT )
   END_RUNG
   RUNG wire#powerrail
      Contact( "LTLP_HMIProInterfaceData".pLamptest )
   END_RUNG wire#w1
   // the same network as SCL:
   #RED_LIGHT := #SAFETY_DOOR.OPEN_OR_UNLOCKED OR "LTLP_HMIProInterfaceData".pLamptest;
END_REGION

REGION Network 38: GREEN LIGHT OUTPUT
   RUNG wire#powerrail
      Contact( #SAFETY_DOOR.CLOSED_AND_LOCKED )
      wire#w1
      Coil( #GREEN_LIGHT )
   END_RUNG
   RUNG wire#powerrail
      Contact( "LTLP_HMIProInterfaceData".pLamptest )
   END_RUNG wire#w1
   // the same network as SCL:
   #GREEN_LIGHT := #SAFETY_DOOR.CLOSED_AND_LOCKED OR "LTLP_HMIProInterfaceData".pLamptest;
END_REGION
END_FUNCTION_BLOCK
